FUNCTION_BLOCK SignalStatusLampComponent_t
VAR_INPUT
END_VAR
VAR_OUTPUT
END_VAR
VAR
	_SignalStatusLamp AT %Q* : BOOL;
	_active : BOOL := FALSE;
	_signalStatusBlink : FB_BA_Blink;
	_blinkerActive : BOOL := FALSE;
	
	_timeOnMS : UDINT;
	_timeOffMS : UDINT;
	
END_VAR

METHOD setStatus : BOOL
VAR_INPUT
	active : BOOL;
	blinking : BOOL := FALSE;
	timeOnMS : UDINT := 100;
	timeOffMS : UDINT := 100;
	
END_VAR
	_active := active;
	_blinkerActive := blinking;
	
	_timeOnMS := timeOnMS;
	_timeOffMS := timeOffMS;
	
	_signalStatusBlink.udiTiOff := timeOffMS;
	_signalStatusBlink.udiTiOn := timeOnMS;
	_signalStatusBlink.bEn := blinking;
END_METHOD

METHOD update : BOOL
VAR_INPUT
END_VAR
_signalStatusBlink();
IF _blinkerActive AND _active THEN 
	_signalStatusBlink.bEn := TRUE;
	_SignalStatusLamp := _signalStatusBlink.bQ;
ELSE 		
	_SignalStatusLamp := _active;
END_IF
END_METHOD

END_FUNCTION_BLOCK

(* stored: Version 1.1.0.1
   POU SignalStatusLampComponent_t: Id {2a0ba243-e24e-47c8-80ba-755d4e515aa5}, SpecialFunc None
   Method setStatus: Id {5e996e2b-7b52-4034-a2af-a9c2690ef38e}
   Method update: Id {1d22d2ea-caad-4ff3-be49-48b5b1fbe736} *)
